{attribute 'qualified_only'}
{attribute 'strict'}
{attribute 'to_string'}
TYPE eErrorReactions :
(
	RESTART := 0,
	ADVANCE := 1,
	CANCEL := 2,
	HOLD :=3
);
END_TYPE

(* stored: Version 1.1.0.1
   DUT eErrorReactions: Id {36d7b298-a784-4157-a495-73a82589c88d} *)
